TYPE ST_SL_Parameter :
STRUCT
	Zeit_Stellen1			: DINT;
	Zeit_Stellen0			: DINT;

	AutoQuittierung			: BOOL;
END_STRUCT
END_TYPE

(* stored: Version 1.1.0.1, ProductVersion 3.1.4024.9
   DUT ST_SL_Parameter: Id {c0877f61-46e9-4587-a16e-ef20c9d361fb} *)
